(* PLC project Test, D OpenPLC 1.0 *)
(* stored: creationDateTime 2018-09-26T00:48:44, modificationDateTime 2018-10-02T13:57:19 *)

PROGRAM Test_Program
  VAR
    ESP0 AT %QX0.0 : BOOL;
  END_VAR
  VAR
    TMP : BOOL;
  END_VAR
  VAR
    ESP1 AT %QX0.1 : BOOL;
  END_VAR
  VAR
    TON1 : TON;
    TON2 : TON;
  END_VAR

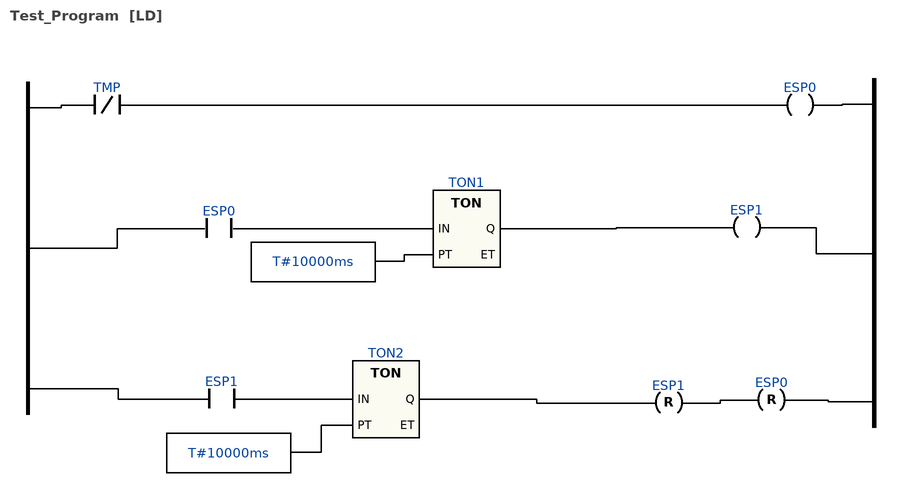
(* LD diagram, written out as Structured Text *)
ESP0 := NOT TMP;
TON1(IN := ESP0, PT := T#10000ms);
ESP1 := TON1.Q;
TON2(IN := ESP1, PT := T#10000ms);
IF TON2.Q THEN ESP1 := FALSE; END_IF;
IF TON2.Q THEN ESP0 := FALSE; END_IF;
END_PROGRAM

CONFIGURATION Config0
  RESOURCE Res0 ON PLC
    TASK MyTask(INTERVAL := T#50ms, PRIORITY := 0);
    PROGRAM instance0 WITH MyTask : Test_Program;
  END_RESOURCE
END_CONFIGURATION
